(* Visualisation PLC_VISU
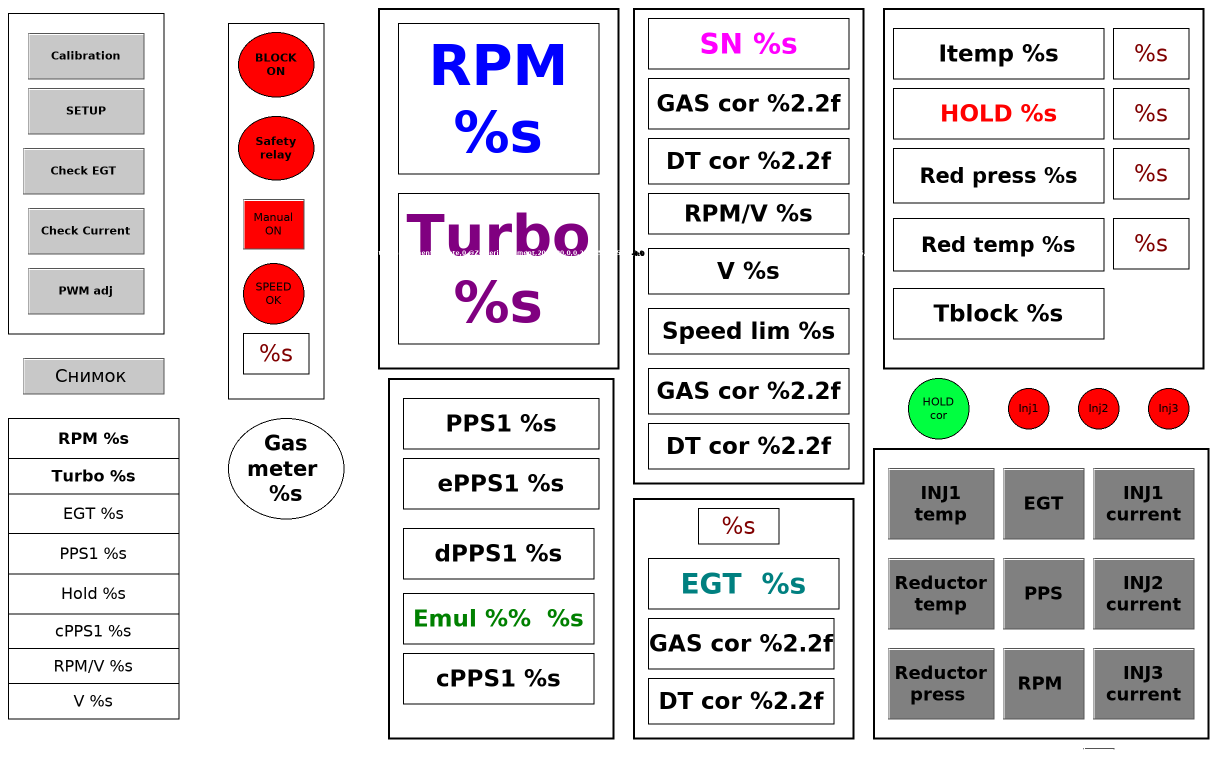
button at (1015,650)-(1096,721): text "RPM"; toggles .Err_RPM
button at (1015,470)-(1096,541): text "EGT"; toggles .Err_EGT
button at (900,560)-(1006,631): text "Reductor / temp"; toggles .Err_Reductor_temp
button at (900,650)-(1006,721): text "Reductor / press"; shows .Reductor_press; toggles .Err_Reductor_press
button at (1105,470)-(1206,541): text "INJ1 / current"; toggles .Err_Inj1
button at (1105,560)-(1206,631): text "INJ2 / current"; toggles .Err_Inj2
button at (900,470)-(1006,541): text "INJ1 / temp"; toggles .Err_Inj_temp
button at (1015,560)-(1096,631): text "PPS"; toggles .Err_PPS
button at (1105,650)-(1206,721): text "INJ3 / current"; toggles .Err_Inj3
ellipse at (1020,390)-(1061,431): text "Inj1"; alarm colour if .Flag_Inj1_ON
ellipse at (1090,390)-(1131,431): text "Inj2"; alarm colour if .Flag_Inj2_ON
ellipse at (1160,390)-(1201,431): text "Inj3"; alarm colour if .Flag_Inj3_ON
ellipse at (920,380)-(981,441): text "HOLD / cor"; alarm colour if .Flag_Inj_PWM_cor
group at (390,10)-(631,371)
  group at (10,210)-(11,211)
    rectangle at (0,0)-(1,1): text "{ExtendedElement},Visu\ElementDLL.ete,0,@Zeigerinstrument,200,180,0,0,255,255,255,0,,,%.1f,0,1,1,1,2,-4,4,0,0,0,0,0,0,0,-13,16,700,Arial,1,2,4000,5500,255,255,128,5500,6000,255,0,0,"
    rectangle at (1,92)-(23,108): text "-4.0"
    rectangle at (27,30)-(49,46): text "-2.0"
    rectangle at (91,4)-(109,20): text "0.0"
    rectangle at (153,30)-(171,46): text "2.0"
    rectangle at (179,92)-(197,108): text "4.0"
  rounded rectangle at (20,185)-(221,336): text "Turbo / %s"; shows .Turbo_pressure
  rounded rectangle at (20,15)-(221,166): text "RPM / %s"; shows .RPM
group at (650,255)-(651,256)
  rectangle at (0,0)-(1,1): text "{ExtendedElement},Visu\ElementDLL.ete,0,@Zeigerinstrument,200,180,0,0,255,255,255,0,,,%.1f,0,1,1,1,2,-4,4,0,0,0,0,0,0,0,-13,16,700,Arial,1,2,4000,5500,255,255,128,5500,6000,255,0,0,"
  rectangle at (1,92)-(23,108): text "-4.0"
  rectangle at (27,30)-(49,46): text "-2.0"
  rectangle at (91,4)-(109,20): text "0.0"
  rectangle at (153,30)-(171,46): text "2.0"
  rectangle at (179,92)-(197,108): text "4.0"
rounded rectangle at (660,195)-(861,236): text "RPM/V %s"; shows .Load
rounded rectangle at (660,250)-(861,296): text "V %s"; shows .Speed
rounded rectangle at (660,20)-(861,71): text "SN %s"; shows .Speed_number
rounded rectangle at (660,80)-(861,131): text "GAS cor %2.2f"; shows Act_control.Gas_cor
rounded rectangle at (660,140)-(861,186): text "DT cor %2.2f"; shows Act_control.Diesel_cor
ellipse at (240,420)-(356,521): text "Gas / meter / %s"; shows .Gas_meter
group at (400,380)-(626,741)
  rounded rectangle at (15,20)-(211,71): text "PPS1 %s"; shows .PPS1
  rounded rectangle at (15,80)-(211,131): text "ePPS1 %s"; shows .PPS1_emul
  rounded rectangle at (15,275)-(206,326): text "cPPS1 %s"; shows .cPPS1_emul
  rounded rectangle at (15,150)-(206,201): text "dPPS1 %s"; shows .PPS1-.PPS1_emul
  rounded rectangle at (15,215)-(206,266): text "Emul %%  %s"; shows 100-((.PPS1_emul-.p.PPS_table[1])*100)/(.PPS1-.p.PPS_table[1])
group at (895,10)-(1216,371)
  rounded rectangle at (10,210)-(221,263): text "Red temp %s"; shows .Reductor_temp
  rounded rectangle at (10,80)-(221,131): text "HOLD %s"; shows .HOLD_time
  rounded rectangle at (10,140)-(221,195): text "Red press %s"; shows .Reductor_press
  rounded rectangle at (10,20)-(221,71): text "Itemp %s"; shows .Injector_temp
  rounded rectangle at (10,280)-(221,331): text "Tblock %s"; shows .gs16_TempBoard
  rectangle at (230,20)-(306,71): text "%s"; shows .p.Inj_temp_max
  rectangle at (230,80)-(306,131): text "%s"; shows .p.Inj_MAX_hold_time/4
  rectangle at (230,140)-(306,191): text "%s"; shows .p.Min_Reductor_press
  rectangle at (230,210)-(306,261): text "%s"; shows .p.Reductor_temp_work
rounded rectangle at (660,310)-(861,356): text "Speed lim %s"; shows .p.Speed_table[12]
rounded rectangle at (660,370)-(861,416): text "GAS cor %2.2f"; shows Act_control.Gas_Speed_cor
rounded rectangle at (660,425)-(861,471): text "DT cor %2.2f"; shows Act_control.Diesel_Speed_cor
button at (40,270)-(156,316): text "PWM adj"; opens PWM_adjustment
button at (40,90)-(156,136): text "SETUP"; opens SETUP
button at (40,210)-(156,256): text "Check Current"; opens CHECK_CURRENT
button at (35,150)-(156,196): text "Check EGT"; opens CHECK_EGT
button at (40,35)-(156,81): text "Calibration"; opens CALIBRATION
group at (240,25)-(336,401)
  ellipse at (10,93)-(86,157): text "Safety / relay"; alarm colour if .gq_Relay
  ellipse at (10,9)-(86,74): text "BLOCK / ON"; alarm colour if .Flag_ECU_ON
  button at (15,176)-(76,226): text "Manual / ON"; toggles .Flag_ECU_ON_VISU
  ellipse at (15,240)-(76,301): text "SPEED / OK"; alarm colour if Get_RPM_speed.Flag_speed_OK
  rectangle at (15,310)-(81,351): text "%s"; shows .p.Speed_limit
rounded rectangle at (660,560)-(851,611): text "EGT  %s"; shows .EGT
rounded rectangle at (660,620)-(846,671): text "GAS cor %2.2f"; shows Act_control.Gas_EGT_cor
rounded rectangle at (660,680)-(846,726): text "DT cor %2.2f"; shows Act_control.Diesel_EGT_cor
rectangle at (710,510)-(791,546): text "%s"; shows .p.EGT_max
rectangle at (20,615)-(191,651): text "cPPS1 %s"; shows .f.cPPS1_emul
button at (35,360)-(176,396): text "Снимок"; taps DFPRS_Change_Cal_Table.Flag_frozen; tooltip Сделать снимок переменных можно нажав ПРОБЕЛ
rectangle at (20,495)-(191,536): text "EGT %s"; shows .f.EGT
rectangle at (20,575)-(191,616): text "Hold %s"; shows .f.Hold_time
rectangle at (20,650)-(191,686): text "RPM/V %s"; shows .f.Load
rectangle at (20,535)-(191,576): text "PPS1 %s"; shows .f.PPS1
rectangle at (20,420)-(191,461): text "RPM %s"; shows .f.RPM
rectangle at (20,685)-(191,721): text "V %s"; shows .f.Speed
rectangle at (20,460)-(191,496): text "Turbo %s"; shows .f.Turbo
35 more shapes without text or variables
*)

(* Visualisation PWM_ADJUSTMENT
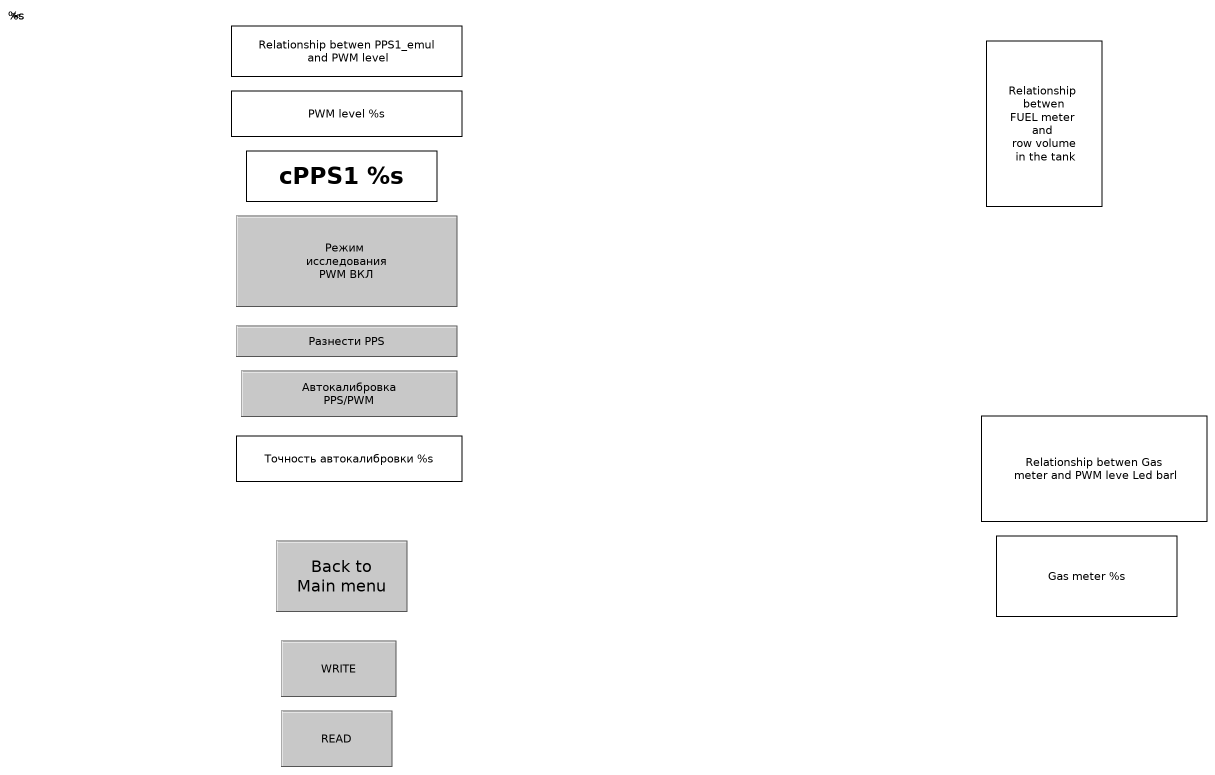
button at (220,200)-(441,291): text "Режим / исследования / PWM ВКЛ"; toggles .Flag_PWM_researh; tooltip Условия включения - нажата Кнопка "ВКЛ Блок" и прогрет редуктор
rounded rectangle at (215,10)-(446,61): text "Relationship betwen PPS1_emul / and PWM level"
rounded rectangle at (215,75)-(446,121): text "PWM level %s"; shows Act_control.PPS_PWM_manual; editable
rectangle at (0,0)-(0,0): text "%s"; shows p.PPS1_emul_PWM[INDEX]; editable
rectangle at (0,0)-(0,0): text "%s"; shows p.PPS_table[INDEX]; editable
rounded rectangle at (230,135)-(421,186): text "cPPS1 %s"; shows .cPPS1_emul
button at (260,525)-(391,596): text "Back to / Main menu"; opens PLC_VISU
rounded rectangle at (970,25)-(1086,191): text "Relationship / betwen / FUEL meter / and / row volume / in the tank"
rounded rectangle at (965,400)-(1191,506): text "Relationship betwen Gas / meter and PWM leve Led barl"
rounded rectangle at (980,520)-(1161,601): text "Gas meter %s"; shows .Gas_meter
button at (220,310)-(441,341): text "Разнести PPS"; taps DFPRS_Change_Cal_Table.Flag_PPS_raznoska; runs 222; tooltip Введите наименьшее и наибольшее значение PPS и нажьмите кнопку, остальные значения будут полученны линейной интерполяцией
button at (225,355)-(441,401): text "Автокалибровка / PPS/PWM"; toggles .Flag_PPS_auto_cal; runs 222; tooltip Условия включения - нажата Кнопка "ВКЛ Блок" и прогрет редуктор
rectangle at (0,0)-(0,0): text "%s"; shows p.LED_BAR_PWM[INDEX]; editable
rectangle at (0,0)-(0,0): text "%s"; shows p.Gas_meter_volume[INDEX]; editable
button at (265,625)-(380,681): text "WRITE"; taps DFPRS_Change_Cal_Table.Write_cal
button at (265,695)-(376,751): text "READ"; taps DFPRS_Change_Cal_Table.Read_cal
rounded rectangle at (220,420)-(446,466): text "Точность автокалибровки %s"; shows Get_cPPS.Precision; tooltip Чем точнее, тем медленнее. Может иметь значения от 1.000 до 60.000; editable
*)

(* Visualisation SETUP
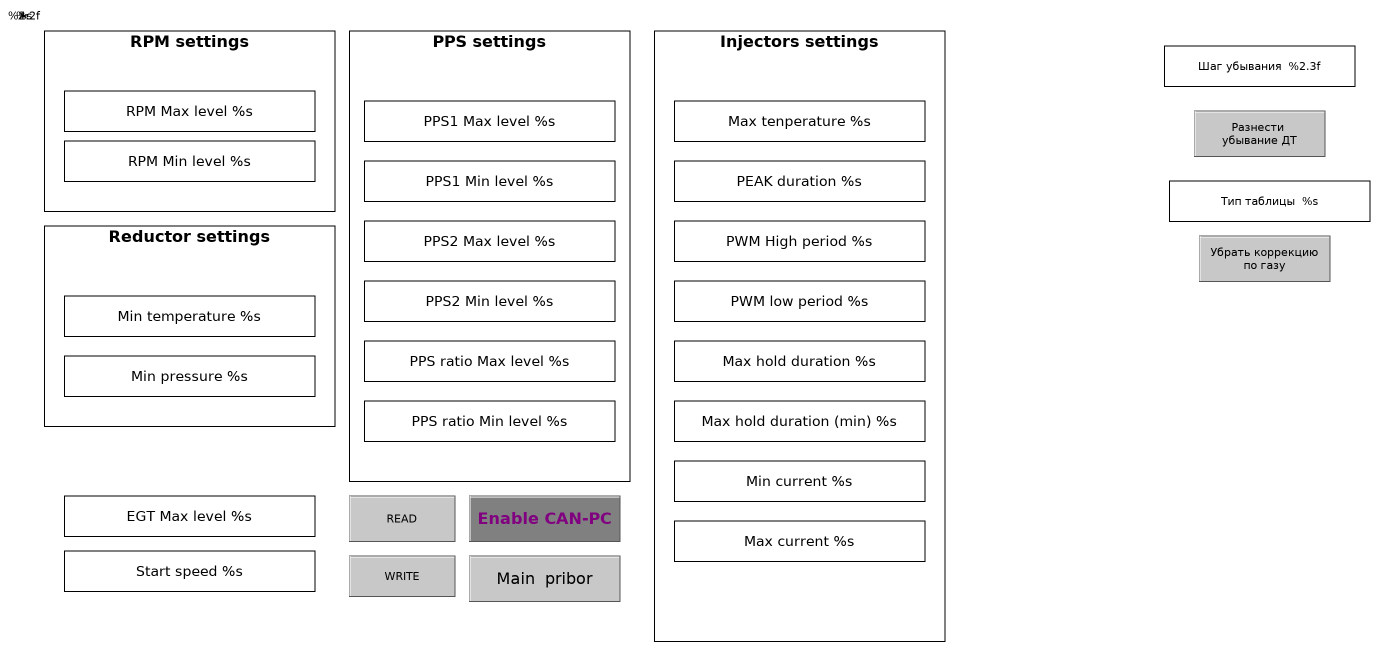
rounded rectangle at (20,210)-(311,411): text "Reductor settings"
rounded rectangle at (20,15)-(311,196): text "RPM settings"
button at (445,480)-(596,526): text "Enable CAN-PC"; toggles .Flag_CAN
rounded rectangle at (40,480)-(291,521): text "EGT Max level %s"; shows .p.EGT_max; editable
button at (325,480)-(431,526): text "READ"; taps DFPRS_Change_Cal_Table.Read_cal
button at (325,540)-(431,581): text "WRITE"; taps DFPRS_Change_Cal_Table.Write_cal
button at (445,540)-(596,586): text "Main  pribor"; opens PLC_VISU
rounded rectangle at (40,75)-(291,116): text "RPM Max level %s"; shows .p.RPM_max; editable
rounded rectangle at (40,125)-(291,166): text "RPM Min level %s"; shows .p.RPM_min; editable
rounded rectangle at (40,280)-(291,321): text "Min temperature %s"; shows .p.Reductor_temp_work; editable
rounded rectangle at (40,340)-(291,381): text "Min pressure %s"; shows .p.Min_Reductor_press; editable
rounded rectangle at (325,15)-(606,466): text "PPS settings"
rounded rectangle at (340,85)-(591,126): text "PPS1 Max level %s"; shows .p.PPS1_max; editable
rounded rectangle at (340,145)-(591,186): text "PPS1 Min level %s"; shows .p.PPS1_min; editable
rounded rectangle at (340,205)-(591,246): text "PPS2 Max level %s"; shows .p.PPS2_max; editable
rounded rectangle at (340,265)-(591,306): text "PPS2 Min level %s"; shows .p.PPS2_min; editable
rounded rectangle at (340,325)-(591,366): text "PPS ratio Max level %s"; shows .p.PPS_ratio_max; editable
rounded rectangle at (340,385)-(591,426): text "PPS ratio Min level %s"; shows .p.PPS_ratio_min; editable
rounded rectangle at (630,15)-(921,626): text "Injectors settings"; tooltip Значения настроек для инжекторов надо менять очень осторожно. И хорошо представлять себя последствия.
rounded rectangle at (650,325)-(901,366): text "Max hold duration %s"; shows .p.Inj_MAX_hold_time; tooltip Абсолютное ограничение максимальной длительности тока удержания. Задается в циклах по 250 мкс. HOLD 1 мс =4*250 мкс; editable
rounded rectangle at (650,385)-(901,426): text "Max hold duration (min) %s"; shows .p.Inj_MAX_hold_time_min; tooltip Ограничение максимальной длительности тока удержания для первых трех значений RPM и Turbo Задается в циклах по 250 мкс. HOLD 1 мс =4*250 мкс; editable
rounded rectangle at (650,265)-(901,306): text "PWM low period %s"; shows .p.Inj_Low_period; tooltip Задание скважности PWM форсунок ( соотношение кол-ва ЦИКЛОВ низкого сигнала к одному ВЫСОКОМУ циклу ), подбирается имперически по условию соблюдения уровня холдового тока на форсунке; editable
rounded rectangle at (650,205)-(901,246): text "PWM High period %s"; shows .p.Inj_High_period; tooltip Задание скважности PWM форсунок ( соотношение кол-ва ЦИКЛОВ низкого сигнала к одному ВЫСОКОМУ циклу ), подбирается имперически по условию соблюдения уровня холдового тока на форсунке; editable
rounded rectangle at (650,145)-(901,186): text "PEAK duration %s"; shows .p.Inj_peak_curent_cycle; tooltip Количество циклов по 250 мкс для генерирования пикового импульса открытия форсунки; editable
rounded rectangle at (650,85)-(901,126): text "Max tenperature %s"; shows .p.Inj_temp_max; tooltip Максимальный ток в микроамперах, протекающий через терморезистор на рейке; editable
rounded rectangle at (650,445)-(901,486): text "Min current %s"; shows .p.Min_inj_current; tooltip Минимальный длительный ток через форсунки; editable
rounded rectangle at (650,505)-(901,546): text "Max current %s"; shows .p.Max_inj_current; tooltip Максимальный длительный ток через форсунки; editable
rounded rectangle at (40,535)-(291,576): text "Start speed %s"; shows .p.Speed_limit; editable
rectangle at (0,0)-(0,0): text "%s"; shows p.Speed_table[INDEX]; editable
rectangle at (0,0)-(0,0): text "%s"; shows p.GAS_Speed_table[INDEX]; editable
rectangle at (0,0)-(0,0): text "%2.2f"; shows p.DIESEL_Speed_table[INDEX]; editable
rounded rectangle at (1140,30)-(1331,71): text "Шаг убывания  %2.3f"; shows DFPRS_Change_Cal_Table.Speed_limit_step; tooltip Максимальный ток в микроамперах, протекающий через терморезистор на рейке; editable
button at (1170,95)-(1301,141): text "Разнести / убывание ДТ"; taps DFPRS_Change_Cal_Table.Flag_speed_limit_raznoska; tooltip Что бы заполнить 1 ( отменить корректировку ) введите Шаг убывания=0
rectangle at (0,0)-(0,0): text "%s"; shows p.Load_table[INDEX]; editable
rectangle at (0,0)-(0,0): text "%s"; shows p.GAS_Load_table[INDEX]; editable
rectangle at (0,0)-(0,0): text "%s"; shows p.DIESEL_Load_table[INDEX]; editable
rounded rectangle at (1145,165)-(1346,206): text "Тип таблицы  %s"; shows DFPRS_Change_Cal_Table.Cor_type; tooltip Выбор типа корректировочной таблицы для разноски убывания ДТ V=ограничитель скорости SN=кореектировка по передаче EGT=корректировка по EGT; editable
rectangle at (0,0)-(0,0): text "%s"; shows p.EGT_table[INDEX]; editable
rectangle at (0,0)-(0,0): text "%s"; shows p.GAS_EGT_table[INDEX]; editable
rectangle at (0,0)-(0,0): text "%s"; shows p.DIESEL_EGT_table[INDEX]; editable
button at (1175,220)-(1306,266): text "Убрать коррекцию / по газу"; taps DFPRS_Change_Cal_Table.Flag_gas_cor_raznoska; tooltip Что бы заполнить 1 ( отменить корректировку ) введите Шаг убывания=0
*)
